(* CODESYS project Esclavo_funciona.project

Project tree, tasks and I/O mapping:
  PLC_AC500_V3 : PM5630-2ETH, ABB AG, order no. 1SAPx31000R0278, version 3.5.0.0
    application Application
      libraries: Util, * (System)
      task Task (cyclic, interval t#10ms, priority 15, watchdog t#20ms x 1) calls PLC_PRG
      CheckConfigurationObject
      program PLC_PRG [ST]
      POUS/
      Diagnosis/
        text list Diag_IO_Bus
        text list Diag_S500_IO_Bus
        text list Diag_V3_PLC
      global variables GVL
    IO_Bus : Bus de E/S, ABB AG, version 3.5.0.0
      DC532 : DC532, ABB AG, order no. 1SAPx40100R0001, version 3.5.0.0
          input  verde : BOOL  // Digital inputs I0 - I7.Digital input I0
          input  verde2 : BOOL  // Digital inputs I0 - I7.Digital input I1
          output salida1 : BOOL  // Digital outputs C16 - C23.Digital output C16
          output salida2 : BOOL  // Digital outputs C16 - C23.Digital output C17
          unmapped channels: Input0, Input1, Input2, Output0, Output1, Digital inputs I0 - I7, Digital inputs I8 - I15, Digital inputs C16 - C23, Digital inputs C24 - C31, Digital outputs C16 - C23, Digital outputs C24 - C31, Digital inputs I0 - I7, Digital inputs I8 - I15, Digital inputs C16 - C23, Digital inputs C24 - C31, Fast counter input, Digital outputs C16 - C23, Digital outputs C24 - C31, Fast counter output, Digital inputs I0 - I7, Digital inputs I8 - I15, Digital inputs C16 - C23, Digital inputs C24 - C31, Digital outputs C16 - C23, Digital outputs C24 - C31
      AX521 : AX521, ABB AG, order no. 1SAPx50100R0001, version 3.5.0.0
          input  Potenciometro : INT  // Analog input I0+
          unmapped channels: Input0, Output0, Analog input I0+, Analog input I1+, Analog input I2+, Analog input I3+, Analog output O0+, Analog output O1+, Analog output O2+, Analog output O3+, Analog input I1+, Analog input I2+, Analog input I3+, Analog output O0+, Analog output O1+, Analog output O2+, Analog output O3+, Analog input I0+, Analog input I1+, Analog input I2+, Analog input I3+, Analog output O0+, Analog output O1+, Analog output O2+, Analog output O3+
    Interfaces : Interfaces, ABB AG, version 3.5.0.0
      COM_1 : COM 1, ABB AG, version 3.5.0.0
        Modbus_RTU_Server : Servidor RTU Modbus, ABB AG, version 3.5.0.0
      CAN
      Ethernet : Ethernet, ABB AG, version 3.5.0.0
        ETH1 : IP Settings, ABB AG, version 3.5.0.0
          NetConfig : Configuración de red, ABB AG, version 3.5.0.0
        ETH2 : IP Settings, ABB AG, version 3.5.0.0
          NetConfig_1 : Configuración de red, ABB AG, version 3.5.0.0
        Protocols : Protocolos cliente, ABB AG, version 3.5.0.0
    Extension_Bus : Bus de ampliación, ABB AG, version 3.5.0.0
      Slot_1
      Slot_2
*)

// PLC_AC500_V3/Application/GVL
{attribute 'qualified_only'}
VAR_GLOBAL
	ILI : WORD;
END_VAR

// PLC_AC500_V3/Application/PLC_PRG
PROGRAM PLC_PRG
VAR
	data AT %MW2: WORD;
END_VAR

data := TO_WORD((Potenciometro * 0.00180584)*163.84);

END_PROGRAM

(* text list Diag_IO_Bus (id | default | en)
  Err_1037 | Test error | Test error
  Err_12 | Test pulse error ->  Check wiring and sensor | Test pulse error ->  Check wiring and sensor
  Err_13 | Test pulse cross-talk error ->  Check wiring and sensor. If this error persists, replace I/O module. Contact ABB technical support. | Test pulse cross-talk error ->  Check wiring and sensor. If this error persists, replace I/O module. Contact ABB technical support.
  Err_16128 | Failed Max Wait Run | Failed Max Wait Run
  Err_16129 | Critical Error, see log | Critical Error, see log
  Err_16130 | Fatal Error, see log | Fatal Error, see log
  Err_16131 | Timeout -> Replace I/O module | Timeout -> Replace I/O module
  Err_16133 | Output data size mismatch | Output data size mismatch
  Err_16134 | Input data size mismatch | Input data size mismatch
  Err_16137 | Overflow diagnosis buffer -> Restart | Overflow diagnosis buffer -> Restart
  Err_16138 | Non-safety I/O: Voltage overflow on outputs (above UP3 level),  Safety I/O: Process voltage too high -> Check terminals/ check process voltage | Non-safety I/O: Voltage overflow on outputs (above UP3 level),  Safety I/O: Process voltage too high -> Check terminals/ check process voltage
  Err_16139 | Process voltage UP or UP3 too low -> Check process voltage | Process voltage UP or UP3 too low -> Check process voltage
  Err_16145 | Error setting parameters | Error setting parameters
  Err_16146 | Plausibility check failed (iParameter) ->  Check configuration | Plausibility check failed (iParameter) ->  Check configuration
  Err_16147 | Checksum error ->  Non-safety I/O: Replace I/O module. Safety I/O: Check safety configuration and CRCs for I- and F-Parameters. | Checksum error ->  Non-safety I/O: Replace I/O module. Safety I/O: Check safety configuration and CRCs for I- and F-Parameters.
  Err_16148 | PROFIsafe communication error ->  Restart I/O module. If this error persists, contact ABB technical support. | PROFIsafe communication error ->  Restart I/O module. If this error persists, contact ABB technical support.
  Err_16149 | No module data | No module data
  Err_16153 | PROFIsafe watchdog timed out ->  Restart I/O module. If this error persists, increase PROFIsafe watchdog time. | PROFIsafe watchdog timed out ->  Restart I/O module. If this error persists, increase PROFIsafe watchdog time.
  Err_16154 | Size of parameters excpeted by module differs from size provided by configuration ->  Check master or configuration | Size of parameters excpeted by module differs from size provided by configuration ->  Check master or configuration
  Err_16156 | F-Parameter configuration and address switch value do not match ->  Check I/O module F-Parameter configuration and module address switch value. | F-Parameter configuration and address switch value do not match ->  Check I/O module F-Parameter configuration and module address switch value.
  Err_16158 | Type of present module does not match configuration | Type of present module does not match configuration
  Err_16159 | Configured number of modules differs from found ones | Configured number of modules differs from found ones
  Err_16160 | At least one module failed during configuration | At least one module failed during configuration
  Err_16164 | Internal data exchange failure -> Replace I/O module | Internal data exchange failure -> Replace I/O module
  Err_16168 | Different hard-/firmware versions in the module -> Replace I/O module | Different hard-/firmware versions in the module -> Replace I/O module
  Err_16171 | Internal error ->  Replace I/O module | Internal error ->  Replace I/O module
  Err_16172 | Has not passed factory test | Has not passed factory test
  Err_16173 | No process voltage UP or UP3 -> Check process voltage | No process voltage UP or UP3 -> Check process voltage
  Err_16175 | Sensor voltage too low | Sensor voltage too low
  Err_16194 | Fatal error, not running any more | Fatal error, not running any more
  Err_16246 | Failed to start the parameterization of modules | Failed to start the parameterization of modules
  Err_16247 | Failed setting parameters | Failed setting parameters
  Err_16248 | Failed setting expected module | Failed setting expected module
  Err_16254 | Size of parameters excpeted by module differs from size provided by configuration | Size of parameters excpeted by module differs from size provided by configuration
  Err_18 | Test error | Test error
  Err_25 | Stuck-at error ->  Check I/O module wiring. Restart I/O module, if needed. If this error persists, replace I/O module. | Stuck-at error ->  Check I/O module wiring. Restart I/O module, if needed. If this error persists, replace I/O module.
  Err_257 | Wrong measurement, false temperature at the compensation channel | Wrong measurement, false temperature at the compensation channel
  Err_258 | AI531: Wrong measurement; potential difference is too high; CD522: PWM duty cycle out of duty area | AI531: Wrong measurement; potential difference is too high; CD522: PWM duty cycle out of duty area
  Err_260 | Measurement overflow ->  Check channel wiring and sensor power supply | Measurement overflow ->  Check channel wiring and sensor power supply
  Err_263 | Measurement underflow ->  Check channel wiring and sensor power supply | Measurement underflow ->  Check channel wiring and sensor power supply
  Err_266 | Short-circuit and cut wire or "out of range" | Short-circuit and cut wire or "out of range"
  Err_267 | Output/process voltage to small/low | Output/process voltage to small/low
  Err_273 | Test error | Test error
  Err_28 | Cross-talk error ->  Check I/O module wiring. Restart I/O module, if needed. If this error persists, replace I/O module. | Cross-talk error ->  Check I/O module wiring. Restart I/O module, if needed. If this error persists, replace I/O module.
  Err_3 | Discrepancy time expired ->  Check discrepancy time value, channel wiring and sensor. | Discrepancy time expired ->  Check discrepancy time value, channel wiring and sensor.
  Err_303 | Short-circuit at the analog input -> Check channel wiring | Short-circuit at the analog input -> Check channel wiring
  Err_304 | Analog value overflow or broken wire at an analog input -> Check value or check terminals | Analog value overflow or broken wire at an analog input -> Check value or check terminals
  Err_311 | Value difference too high ->  Adjust tolerance window for channels. Check channel wiring and sensor configuration. | Value difference too high ->  Adjust tolerance window for channels. Check channel wiring and sensor configuration.
  Err_524 | Stuck-at error | Stuck-at error
  Err_525 | Readback error ->  Check I/O module wiring. Restart I/O module, if needed. If this error persists, replace I/O module. | Readback error ->  Check I/O module wiring. Restart I/O module, if needed. If this error persists, replace I/O module.
  Err_530 | Class 3: Cross-talk error; Class 4: Internal fuse at 0V is defect. 0V not conected with GND. ->  Check I/O module wiring. Restart I/O module, if needed. If this error persists, replace I/O module. | Class 3: Cross-talk error; Class 4: Internal fuse at 0V is defect. 0V not conected with GND. ->  Check I/O module wiring. Restart I/O module, if needed. If this error persists, replace I/O module.
  Err_540 | Test error | Test error
  Err_555 | Internal error | Internal error
  Err_559 | Short-circuit at the digital output -> Check channel wiring | Short-circuit at the digital output -> Check channel wiring
  Err_775 | Measurement underflow at analog input ->  Check channel wiring | Measurement underflow at analog input ->  Check channel wiring
  Err_796 | Different configuration | Different configuration
  Err_8480 | Not supported protocol variant | Not supported protocol variant
  Err_8482 | Class 2: Timeout while initializing; Class 4: Timeout while waiting for ready status | Class 2: Timeout while initializing; Class 4: Timeout while waiting for ready status
  Err_8483 | Timeout during parameterization | Timeout during parameterization
  Err_8707 | PROFIsafe watchdog timed out | PROFIsafe watchdog timed out
  Err_8708 | Overvoltage | Overvoltage
  Err_8711 | Undervoltage | Undervoltage
  Err_8722 | Internal error | Internal error
  Err_8723 | Checksum error has occured in iParameters | Checksum error has occured in iParameters
  Err_8724 | PROFIsafe communication error | PROFIsafe communication error
  Err_8732 | Internal error  | Internal error 
  Err_8747 | Internal runtime error | Internal runtime error
  Err_8961 | Wrong parameter value, check configuration | Wrong parameter value, check configuration
  Err_8979 | Checksum error has occured in iParameter or F-Parameters | Checksum error has occured in iParameter or F-Parameters
  Err_8986 | Invalid configuration -> Check modules and parameterization | Invalid configuration -> Check modules and parameterization
  Err_8988 | F-Parameter configuration and address switch value do not match ->  Check I/O module F-Parameter configuration and module address switch value. | F-Parameter configuration and address switch value do not match ->  Check I/O module F-Parameter configuration and module address switch value.
  Err_9249 | Timeout while waiting for Reset | Timeout while waiting for Reset
  Err_9258 | Breakdown, communication lost | Breakdown, communication lost
  Err_9480 | I/O module removed from HotSwap terminal unit or defective module on HotSwap terminal unit -> Plug I/O module, replace I/O module | I/O module removed from HotSwap terminal unit or defective module on HotSwap terminal unit -> Plug I/O module, replace I/O module
  Err_9500 | Wrong I/O module plugged on HotSwap terminal unit -> Remove wrong I/O module and plug projected I/O module | Wrong I/O module plugged on HotSwap terminal unit -> Remove wrong I/O module and plug projected I/O module
  Err_9514 | No communication with I/O module on HotSwap terminal unit -> Replace I/O module | No communication with I/O module on HotSwap terminal unit -> Replace I/O module
  Err_9526 | I/O module does not support HotSwap functionality -> Power off system and replace I/O module | I/O module does not support HotSwap functionality -> Power off system and replace I/O module
  Err_9736 | HotSwap Terminal Unit required but not found | HotSwap Terminal Unit required but not found
  Err_9764 | Defective HotSwap Terminal Unit | Defective HotSwap Terminal Unit
  Err_9770 | No communication with HotSwap terminal unit -> Restart, if error persists replace terminal unit | No communication with HotSwap terminal unit -> Restart, if error persists replace terminal unit
  Hwd_14 | I/O-Bus | I/O-Bus
  Sub1_ | Module | Module
  Sub2_ | Channel | Channel *)

(* text list Diag_S500_IO_Bus (id | default | en)
  Err_1037 | Test error | Test error
  Err_12 | Test pulse error ->  Check wiring and sensor | Test pulse error ->  Check wiring and sensor
  Err_13 | Test pulse cross-talk error ->  Check wiring and sensor. If this error persists, replace I/O module. Contact ABB technical support. | Test pulse cross-talk error ->  Check wiring and sensor. If this error persists, replace I/O module. Contact ABB technical support.
  Err_16128 | Failed Max Wait Run | Failed Max Wait Run
  Err_16129 | Critical Error, see log | Critical Error, see log
  Err_16130 | Fatal Error, see log | Fatal Error, see log
  Err_16131 | Timeout -> Replace I/O module | Timeout -> Replace I/O module
  Err_16133 | Output data size mismatch | Output data size mismatch
  Err_16134 | Input data size mismatch | Input data size mismatch
  Err_16137 | Overflow diagnosis buffer -> Restart | Overflow diagnosis buffer -> Restart
  Err_16138 | Non-safety I/O: Voltage overflow on outputs (above UP3 level),  Safety I/O: Process voltage too high -> Check terminals/ check process voltage | Non-safety I/O: Voltage overflow on outputs (above UP3 level),  Safety I/O: Process voltage too high -> Check terminals/ check process voltage
  Err_16139 | Process voltage UP or UP3 too low -> Check process voltage | Process voltage UP or UP3 too low -> Check process voltage
  Err_16145 | Error setting parameters | Error setting parameters
  Err_16146 | Plausibility check failed (iParameter) ->  Check configuration | Plausibility check failed (iParameter) ->  Check configuration
  Err_16147 | Checksum error ->  Non-safety I/O: Replace I/O module. Safety I/O: Check safety configuration and CRCs for I- and F-Parameters. | Checksum error ->  Non-safety I/O: Replace I/O module. Safety I/O: Check safety configuration and CRCs for I- and F-Parameters.
  Err_16148 | PROFIsafe communication error ->  Restart I/O module. If this error persists, contact ABB technical support. | PROFIsafe communication error ->  Restart I/O module. If this error persists, contact ABB technical support.
  Err_16149 | No module data | No module data
  Err_16153 | PROFIsafe watchdog timed out ->  Restart I/O module. If this error persists, increase PROFIsafe watchdog time. | PROFIsafe watchdog timed out ->  Restart I/O module. If this error persists, increase PROFIsafe watchdog time.
  Err_16154 | Size of parameters excpeted by module differs from size provided by configuration ->  Check master or configuration | Size of parameters excpeted by module differs from size provided by configuration ->  Check master or configuration
  Err_16156 | F-Parameter configuration and address switch value do not match ->  Check I/O module F-Parameter configuration and module address switch value. | F-Parameter configuration and address switch value do not match ->  Check I/O module F-Parameter configuration and module address switch value.
  Err_16158 | Type of present module does not match configuration | Type of present module does not match configuration
  Err_16159 | Configured number of modules differs from found ones | Configured number of modules differs from found ones
  Err_16160 | At least one module failed during configuration | At least one module failed during configuration
  Err_16164 | Internal data exchange failure -> Replace I/O module | Internal data exchange failure -> Replace I/O module
  Err_16168 | Different hard-/firmware versions in the module -> Replace I/O module | Different hard-/firmware versions in the module -> Replace I/O module
  Err_16171 | Internal error ->  Replace I/O module | Internal error ->  Replace I/O module
  Err_16172 | Has not passed factory test | Has not passed factory test
  Err_16173 | No process voltage UP or UP3 -> Check process voltage | No process voltage UP or UP3 -> Check process voltage
  Err_16175 | Sensor voltage too low | Sensor voltage too low
  Err_16194 | Fatal error, not running any more | Fatal error, not running any more
  Err_16246 | Failed to start the parameterization of modules | Failed to start the parameterization of modules
  Err_16247 | Failed setting parameters | Failed setting parameters
  Err_16248 | Failed setting expected module | Failed setting expected module
  Err_16254 | Size of parameters excpeted by module differs from size provided by configuration | Size of parameters excpeted by module differs from size provided by configuration
  Err_18 | Test error | Test error
  Err_25 | Stuck-at error ->  Check I/O module wiring. Restart I/O module, if needed. If this error persists, replace I/O module. | Stuck-at error ->  Check I/O module wiring. Restart I/O module, if needed. If this error persists, replace I/O module.
  Err_257 | Wrong measurement, false temperature at the compensation channel | Wrong measurement, false temperature at the compensation channel
  Err_258 | AI531: Wrong measurement; potential difference is too high; CD522: PWM duty cycle out of duty area | AI531: Wrong measurement; potential difference is too high; CD522: PWM duty cycle out of duty area
  Err_260 | Measurement overflow ->  Check channel wiring and sensor power supply | Measurement overflow ->  Check channel wiring and sensor power supply
  Err_263 | Measurement underflow ->  Check channel wiring and sensor power supply | Measurement underflow ->  Check channel wiring and sensor power supply
  Err_266 | Short-circuit and cut wire or "out of range" | Short-circuit and cut wire or "out of range"
  Err_267 | Output/process voltage to small/low | Output/process voltage to small/low
  Err_273 | Test error | Test error
  Err_28 | Cross-talk error ->  Check I/O module wiring. Restart I/O module, if needed. If this error persists, replace I/O module. | Cross-talk error ->  Check I/O module wiring. Restart I/O module, if needed. If this error persists, replace I/O module.
  Err_3 | Discrepancy time expired ->  Check discrepancy time value, channel wiring and sensor. | Discrepancy time expired ->  Check discrepancy time value, channel wiring and sensor.
  Err_303 | Short-circuit at the analog input -> Check channel wiring | Short-circuit at the analog input -> Check channel wiring
  Err_304 | Analog value overflow or broken wire at an analog input -> Check value or check terminals | Analog value overflow or broken wire at an analog input -> Check value or check terminals
  Err_311 | Value difference too high ->  Adjust tolerance window for channels. Check channel wiring and sensor configuration. | Value difference too high ->  Adjust tolerance window for channels. Check channel wiring and sensor configuration.
  Err_524 | Stuck-at error | Stuck-at error
  Err_525 | Readback error ->  Check I/O module wiring. Restart I/O module, if needed. If this error persists, replace I/O module. | Readback error ->  Check I/O module wiring. Restart I/O module, if needed. If this error persists, replace I/O module.
  Err_530 | Class 3: Cross-talk error; Class 4: Internal fuse at 0V is defect. 0V not conected with GND. ->  Check I/O module wiring. Restart I/O module, if needed. If this error persists, replace I/O module. | Class 3: Cross-talk error; Class 4: Internal fuse at 0V is defect. 0V not conected with GND. ->  Check I/O module wiring. Restart I/O module, if needed. If this error persists, replace I/O module.
  Err_540 | Test error | Test error
  Err_555 | Internal error | Internal error
  Err_559 | Short-circuit at the digital output -> Check channel wiring | Short-circuit at the digital output -> Check channel wiring
  Err_7_1037 | Test error | Test error
  Err_7_1070 | Externally voltage detected on digital output DC0...DC7 -> Check terminals | Externally voltage detected on digital output DC0...DC7 -> Check terminals
  Err_7_1071 | Short circuit at digital output -> Check terminals | Short circuit at digital output -> Check terminals
  Err_7_16131 | Timeout -> Replace I/O module | Timeout -> Replace I/O module
  Err_7_16137 | Overflow diagnosis buffer -> Restart | Overflow diagnosis buffer -> Restart
  Err_7_16138 | Voltage overflow at outputs (above UP3 level) -> Check terminals / check process supply voltage | Voltage overflow at outputs (above UP3 level) -> Check terminals / check process supply voltage
  Err_7_16139 | Process voltage UP or UP3 too low -> Check process supply voltage | Process voltage UP or UP3 too low -> Check process supply voltage
  Err_7_16145 | No communication with I/O device -> Replace I/O module | No communication with I/O device -> Replace I/O module
  Err_7_16147 | Checksum error -> Replace I/O module | Checksum error -> Replace I/O module
  Err_7_16154 | Parameter error -> Check configuration | Parameter error -> Check configuration
  Err_7_16159 | At least one module does not support failsafe function -> Check modules and parameterization | At least one module does not support failsafe function -> Check modules and parameterization
  Err_7_16160 | Wrong I/O device type on socket -> Replace I/O module / check configuration | Wrong I/O device type on socket -> Replace I/O module / check configuration
  Err_7_16162 | No response during initialization of the I/O module -> Replace I/O module | No response during initialization of the I/O module -> Replace I/O module
  Err_7_16164 | Internal data exchange failure -> Replace I/O module | Internal data exchange failure -> Replace I/O module
  Err_7_16168 | Different hard-/firmware versions in the module -> Replace I/O module | Different hard-/firmware versions in the module -> Replace I/O module
  Err_7_16171 | Internal error -> Replace I/O module | Internal error -> Replace I/O module
  Err_7_16173 | No process voltage UP or UP3 -> Check process voltage | No process voltage UP or UP3 -> Check process voltage
  Err_7_16174 | Voltage feedback on activated digital outputs DO0...DO7 on UP3 -> Check terminals | Voltage feedback on activated digital outputs DO0...DO7 on UP3 -> Check terminals
  Err_7_16175 | Sensor voltage too low | Sensor voltage too low
  Err_7_18 | Test error | Test error
  Err_7_257 | Wrong measurement, false temperature at the compensation channel | Wrong measurement, false temperature at the compensation channel
  Err_7_258 | AI531: Wrong measurement; potential difference is too high; CD522: PWM duty cycle out of duty area | AI531: Wrong measurement; potential difference is too high; CD522: PWM duty cycle out of duty area
  Err_7_260 | Measurement overflow -> Check channel wiring and sensor power supply | Measurement overflow -> Check channel wiring and sensor power supply
  Err_7_263 | Measurement underflow at analog input -> Check channel wiring and sensor power supply | Measurement underflow at analog input -> Check channel wiring and sensor power supply
  Err_7_266 | Short circuit and cut wire or "out of range" | Short circuit and cut wire or "out of range"
  Err_7_267 | Output/process voltage to small/low | Output/process voltage to small/low
  Err_7_273 | Test error | Test error
  Err_7_303 | Short circuit at an analog input -> Check channel wiring | Short circuit at an analog input -> Check channel wiring
  Err_7_304 | Analog value overflow or broken wire at an analog input -> Check value or check terminals | Analog value overflow or broken wire at an analog input -> Check value or check terminals
  Err_7_530 | Internal fuse at 0V is defect. 0V not conected with GND -> Check I/O module wiring. Restart I/O module, if needed. If this error persists, replace I/O module | Internal fuse at 0V is defect. 0V not conected with GND -> Check I/O module wiring. Restart I/O module, if needed. If this error persists, replace I/O module
  Err_7_540 | Test error | Test error
  Err_7_555 | Internal error | Internal error
  Err_7_558 | Externally voltage detected on digital output DO0...DO7 -> Check terminals | Externally voltage detected on digital output DO0...DO7 -> Check terminals
  Err_7_559 | Short circuit at digital output -> Check channel wiring | Short circuit at digital output -> Check channel wiring
  Err_7_772 | Analog value overflow at an analog output -> Check output value | Analog value overflow at an analog output -> Check output value
  Err_7_775 | Analog value underflow at an analog output -> Check output value | Analog value underflow at an analog output -> Check output value
  Err_7_796 | Different configuration | Different configuration
  Err_7_8722 | Internal error | Internal error
  Err_7_8732 | Internal error | Internal error
  Err_7_9480 | I/O module removed from hot swap terminal unit or defective module on hot swap terminal unit -> Plug I/O module, replace I/O module | I/O module removed from hot swap terminal unit or defective module on hot swap terminal unit -> Plug I/O module, replace I/O module
  Err_7_9500 | Wrong I/O module plugged on hot swap terminal unit -> Remove wrong I/O module and plug projected I/O module | Wrong I/O module plugged on hot swap terminal unit -> Remove wrong I/O module and plug projected I/O module
  Err_7_9514 | No communication with I/O module on hot swap terminal unit -> Replace I/O module | No communication with I/O module on hot swap terminal unit -> Replace I/O module
  Err_7_9526 | I/O module does not support hot swap -> Power off system and replace I/O module | I/O module does not support hot swap -> Power off system and replace I/O module
  Err_7_9736 | Hot swap terminal unit required but not found -> Plug hot swap terminal unit | Hot swap terminal unit required but not found -> Plug hot swap terminal unit
  Err_7_9764 | Defective hot swap terminal unit | Defective hot swap terminal unit
  Err_7_9770 | No communication with hot swap terminal unit -> Restart, if error persists replace terminal unit | No communication with hot swap terminal unit -> Restart, if error persists replace terminal unit
  Err_775 | Measurement underflow at analog input ->  Check channel wiring | Measurement underflow at analog input ->  Check channel wiring
  Err_796 | Different configuration | Different configuration
  Err_8480 | Not supported protocol variant | Not supported protocol variant
  Err_8482 | Class 2: Timeout while initializing; Class 4: Timeout while waiting for ready status | Class 2: Timeout while initializing; Class 4: Timeout while waiting for ready status
  Err_8483 | Timeout during parameterization | Timeout during parameterization
  Err_8707 | PROFIsafe watchdog timed out | PROFIsafe watchdog timed out
  Err_8708 | Overvoltage | Overvoltage
  Err_8711 | Undervoltage | Undervoltage
  Err_8722 | Internal error | Internal error
  Err_8723 | Checksum error has occured in iParameters | Checksum error has occured in iParameters
  Err_8724 | PROFIsafe communication error | PROFIsafe communication error
  Err_8732 | Internal error  | Internal error 
  Err_8747 | Internal runtime error | Internal runtime error
  Err_8961 | Wrong parameter value, check configuration | Wrong parameter value, check configuration
  Err_8979 | Checksum error has occured in iParameter or F-Parameters | Checksum error has occured in iParameter or F-Parameters
  Err_8986 | Invalid configuration -> Check modules and parameterization | Invalid configuration -> Check modules and parameterization
  Err_8988 | F-Parameter configuration and address switch value do not match ->  Check I/O module F-Parameter configuration and module address switch value. | F-Parameter configuration and address switch value do not match ->  Check I/O module F-Parameter configuration and module address switch value.
  Err_9249 | Timeout while waiting for Reset | Timeout while waiting for Reset
  Err_9258 | Breakdown, communication lost | Breakdown, communication lost
  Err_9480 | I/O module removed from HotSwap terminal unit or defective module on HotSwap terminal unit -> Plug I/O module, replace I/O module | I/O module removed from HotSwap terminal unit or defective module on HotSwap terminal unit -> Plug I/O module, replace I/O module
  Err_9500 | Wrong I/O module plugged on HotSwap terminal unit -> Remove wrong I/O module and plug projected I/O module | Wrong I/O module plugged on HotSwap terminal unit -> Remove wrong I/O module and plug projected I/O module
  Err_9514 | No communication with I/O module on HotSwap terminal unit -> Replace I/O module | No communication with I/O module on HotSwap terminal unit -> Replace I/O module
  Err_9526 | I/O module does not support HotSwap functionality -> Power off system and replace I/O module | I/O module does not support HotSwap functionality -> Power off system and replace I/O module
  Err_9736 | HotSwap Terminal Unit required but not found | HotSwap Terminal Unit required but not found
  Err_9764 | Defective HotSwap Terminal Unit | Defective HotSwap Terminal Unit
  Err_9770 | No communication with HotSwap terminal unit -> Restart, if error persists replace terminal unit | No communication with HotSwap terminal unit -> Restart, if error persists replace terminal unit
  Hwd_14 | I/O-Bus | I/O-Bus
  Sub1_ | Module | Module
  Sub2_ | Channel | Channel *)

(* text list Diag_V3_PLC (id | default | en)
  Add_570425344 | Unknown reason | Unknown reason
  Add_570425345 | Shutdown of the PLC | Shutdown of the PLC
  Add_570425346 | Reset after having stopped the IEC application | Reset after having stopped the IEC application
  Add_570425347 | Exception occurred | Exception occurred
  Add_570425348 | IEC application stopped by user | IEC application stopped by user
  Add_570425349 | IEC application stopped by function block | IEC application stopped by function block
  Add_570425350 | IEC application will be deleted after the stop | IEC application will be deleted after the stop
  Add_570425351 | IEC application stopped because of debugging | IEC application stopped because of debugging
  Add_570425352 | IEC application stopped because the run stop switch is on stop | IEC application stopped because the run stop switch is on stop
  Add_587202560 | Reset warm | Reset warm
  Add_587202561 | Reset cold | Reset cold
  Add_587202562 | Reset origin | Reset origin
  Add_587202563 | Reset device | Reset device
  Add_637534224 | Software watchdog of IEC task expired | Software watchdog of IEC task expired
  Add_637534225 | Hardware watchdog expired. Global software error | Hardware watchdog expired. Global software error
  Add_637534226 | I/O configuration error | I/O configuration error
  Add_637534227 | Checksum error after program download | Checksum error after program download
  Add_637534228 | Fieldbus error | Fieldbus error
  Add_637534229 | I/O update error | I/O update error
  Add_637534230 | Cycle time exceeded | Cycle time exceeded
  Add_637534231 | Program too large for online change | Program too large for online change
  Add_637534232 | Unresolved external references | Unresolved external references
  Add_637534233 | Download was rejected | Download was rejected
  Add_637534234 | Boot project not loaded because retain variables could not be relocated | Boot project not loaded because retain variables could not be relocated
  Add_637534235 | Boot project not loaded and deleted | Boot project not loaded and deleted
  Add_637534236 | Out of heap memory | Out of heap memory
  Add_637534237 | Retain memory corrupt or cannot be mapped | Retain memory corrupt or cannot be mapped
  Add_637534238 | Boot project could be loaded but caused an exception | Boot project could be loaded but caused an exception
  Add_637534241 | Target of the boot application doesn't match the current target | Target of the boot application doesn't match the current target
  Add_637534242 | Error at scheduling IEC tasks | Error at scheduling IEC tasks
  Add_637534243 | Checksum of downloaded file does not match | Checksum of downloaded file does not match
  Add_637534244 | Retain identity does not match to current boot application program identity | Retain identity does not match to current boot application program identity
  Add_637534245 | IEC task configuration failed | IEC task configuration failed
  Add_637534246 | Application is running on wrong target. Can be used for library protection! | Application is running on wrong target. Can be used for library protection!
  Add_637534288 | Illegal instruction | Illegal instruction
  Add_637534289 | Access violation | Access violation
  Add_637534290 | Privileged instruction | Privileged instruction
  Add_637534292 | Stack overflow | Stack overflow
  Add_637534293 | Invalid disposition | Invalid disposition
  Add_637534294 | Invalid handle | Invalid handle
  Add_637534295 | Guard page | Guard page
  Add_637534296 | Double fault | Double fault
  Add_637534297 | Invalid OpCode | Invalid OpCode
  Add_637534464 | Data type misalignment | Data type misalignment
  Add_637534465 | Array bounds exceeded | Array bounds exceeded
  Add_637534466 | Division by zero | Division by zero
  Add_637534467 | Overflow | Overflow
  Add_637534468 | Non continuable | Non continuable
  Add_637534469 | Processor load watchdog of all IEC tasks detected | Processor load watchdog of all IEC tasks detected
  Add_637534544 | FPU: Unspecified error | FPU: Unspecified error
  Add_637534545 | FPU: Denormalized operand | FPU: Denormalized operand
  Add_637534546 | FPU: Division by zero | FPU: Division by zero
  Add_637534547 | FPU: Inexact result | FPU: Inexact result
  Add_637534548 | FPU: Invalid operation | FPU: Invalid operation
  Add_637534549 | FPU: Overflow | FPU: Overflow
  Add_637534550 | FPU: Stack check | FPU: Stack check
  Add_637534551 | FPU: Underflow | FPU: Underflow
  Add_637534720 | Hardware breakpoint | Hardware breakpoint
  Add_637538320 | Omitted cycle watchdog | Omitted cycle watchdog
  Err_10 | Medium has almost used its complete spare capacity or is already dead, action required | Medium has almost used its complete spare capacity or is already dead, action required
  Err_11 | Type scaling on PLC startup failed | Type scaling on PLC startup failed
  Err_12 | Flash is temporary protected (read only, panic mode) | Flash is temporary protected (read only, panic mode)
  Err_17 | Error setting parameter | Error setting parameter
  Err_18 | At least one not found | At least one not found
  Err_19 | Unable to read at least one value | Unable to read at least one value
  Err_2 | Resource failure | Resource failure
  Err_20 | Invalid value of "Error LED" | Invalid value of "Error LED"
  Err_21 | Invalid value of "Check battery" | Invalid value of "Check battery"
  Err_22 | Error at initialization | Error at initialization
  Err_23 | Wrong version of firmware | Wrong version of firmware
  Err_24 | Invalid value of parameter "Diagnosis, stop on error class" | Invalid value of parameter "Diagnosis, stop on error class"
  Err_25 | Invalid value of parameter "Diagnosis, add Plc name to node name" | Invalid value of parameter "Diagnosis, add Plc name to node name"
  Err_26 | Invalid value of parameter "Reboot at powerfail" | Invalid value of parameter "Reboot at powerfail"
  Err_27 | Failed to set parameter "Reboot at powerfail" | Failed to set parameter "Reboot at powerfail"
  Err_28 | Value of parameter "Missed Cycle Task behaviour" is not in range | Value of parameter "Missed Cycle Task behaviour" is not in range
  Err_29 | Combination of plugged option boards is invalid | Combination of plugged option boards is invalid
  Err_3 | Timeout | Timeout
  Err_30 | Value of parameter "Priority Scheme" is not in range | Value of parameter "Priority Scheme" is not in range
  Err_31 | PLC did not go to RUN mode due to an active error, whose severity exceeds value of parameter 'stop on error class' | PLC did not go to RUN mode due to an active error, whose severity exceeds value of parameter 'stop on error class'
  Err_32 | PLC went to STOP mode due to occurence of an error, whose severity exceeds value of parameter 'stop on error class' | PLC went to STOP mode due to occurence of an error, whose severity exceeds value of parameter 'stop on error class'
  Err_33 | PLC went to RUN mode | PLC went to RUN mode
  Err_34 | PLC went to STOP mode | PLC went to STOP mode
  Err_35 | IEC application has been reset | IEC application has been reset
  Err_36 | Online change of IEC application has been performed | Online change of IEC application has been performed
  Err_37 | Full download of an IEC application has been performed | Full download of an IEC application has been performed
  Err_38 | IEC application caused an exception | IEC application caused an exception
  Err_39 | PLC did not go to RUN mode since reboot has to be performed first | PLC did not go to RUN mode since reboot has to be performed first
  Err_40 | Value of parameter "Reboot on E2" is not in range | Value of parameter "Reboot on E2" is not in range
  Err_41 | PLC went to REBOOT due to occurence of an E2 error | PLC went to REBOOT due to occurence of an E2 error
  Err_42 | No bootproject loaded | No bootproject loaded
  Err_43 | Bootproject loaded | Bootproject loaded
  Err_44 | Loading boot project failed due to failing load of retain data | Loading boot project failed due to failing load of retain data
  Err_45 | Loading boot project failed due to mismatch of retain data | Loading boot project failed due to mismatch of retain data
  Err_46 | Loading boot project failed due to insufficient license for application | Loading boot project failed due to insufficient license for application
  Err_47 | Loading boot project failed due to unspecified reason | Loading boot project failed due to unspecified reason
  Err_48 | Backup failed | Backup failed
  Err_49 | Restore failed | Restore failed
  Err_8 | Empty or missing | Empty or missing
  Err_9 | Medium has used 80% of its spare capacity | Medium has used 80% of its spare capacity
  Hwd_0 | CPU | CPU
  Sub1_0 | CPU | CPU
  Sub1_14 | I/O-Bus | I/O-Bus
  Sub1_19 | Flashdisk | Flashdisk
  Sub1_21 | Display | Display
  Sub1_22 | Battery | Battery
  Sub2_0 | Device | Device
  Sub2_2 | Parameter | Parameter
  Sub2_5 | Index | Index
  Sub2_6 | Application | Application
  Sub4_1 | too big | too big
  Sub4_2 | too small | too small
  Sub4_3 | unequal | unequal
  Sub4_4 | equal | equal *)
